ABB RobotStudio station: roboticcell.rsstnx

Station roboticcell (saved by RobotStudio 23.2.10395.0)
Controller Controller2
  mechanical unit ROB_1: IRB2600_20_165_C_01_2, 6 joints, base frame (0, 0, 0) mm
Layout (positions relative to the parent item):
  - IRB2600_20_165_C_01_2 [mechanism, from %ABB.RobotStudio.Models.IRB2600%\IRB2600_20_165_C_01.rslib] at (0, 0, 0) mm; joint values [0.1279, 0.0673, -0.394, 2.9455, -0.603, -2.0324] (rad or m)
  - 2FGP20_WEB_26012022_3 [graphiccomponentgroup] at (0, 0, 0) mm, rotated rx 0 ry 0 rz 90 deg
    - 108791 [graphiccomponentgroup] at (0, 153, -120.5) mm, rotated rx 90 ry 0 rz 180 deg
      - 108659 [graphiccomponentgroup] at (205, 123, 11.8) mm, rotated rx 90 ry 0 rz 24.4 deg
        - 108790 [part] at (0, 0, 0) mm, rotated rx 180 ry 0 rz 0 deg, size 17 x 14.6 x 17 mm
        - 101019 [part] at (0, -6.3, 0) mm, rotated rx 180 ry 74.5 rz 0 deg, size 40 x 26 x 40 mm
        - 104702_Standard [part] at (0, -27.2, 0) mm, rotated rx 90 ry -9.84 rz 180 deg, size 23.8 x 13 x 23.4 mm
        - 109120 [part] at (0, -11.45, 0) mm, rotated rx 180 ry -25.08 rz 0 deg, size 12.6 x 1.3 x 12.6 mm
      - 108659-1 [graphiccomponentgroup] at (-205, 123, 11.8) mm, rotated rx 90 ry 0 rz 137.17 deg
        - 108790 [part] at (0, 0, 0) mm, rotated rx 180 ry 0 rz 0 deg, size 17 x 14.6 x 17 mm
        - 101019 [part] at (0, -6.3, 0) mm, rotated rx 180 ry 74.5 rz 0 deg, size 40 x 26 x 40 mm
        - 104702_Standard [part] at (0, -27.2, 0) mm, rotated rx 90 ry -9.84 rz 180 deg, size 23.8 x 13 x 23.4 mm
        - 109120 [part] at (0, -11.45, 0) mm, rotated rx 180 ry -25.08 rz 0 deg, size 12.6 x 1.3 x 12.6 mm
      - 108659-2 [graphiccomponentgroup] at (205, 8.5, 11.8) mm, rotated rx 90 ry 0 rz -12.46 deg
        - 108790 [part] at (0, 0, 0) mm, rotated rx 180 ry 0 rz 0 deg, size 17 x 14.6 x 17 mm
        - 101019 [part] at (0, -6.3, 0) mm, rotated rx 180 ry 74.5 rz 0 deg, size 40 x 26 x 40 mm
        - 104702_Standard [part] at (0, -27.2, 0) mm, rotated rx 90 ry -9.84 rz 180 deg, size 23.8 x 13 x 23.4 mm
        - 109120 [part] at (0, -11.45, 0) mm, rotated rx 180 ry -25.08 rz 0 deg, size 12.6 x 1.3 x 12.6 mm
      - 108659-3 [graphiccomponentgroup] at (-205, 8.5, 11.8) mm, rotated rx 90 ry 0 rz 173.2 deg
        - 108790 [part] at (0, 0, 0) mm, rotated rx 180 ry 0 rz 0 deg, size 17 x 14.6 x 17 mm
        - 101019 [part] at (0, -6.3, 0) mm, rotated rx 180 ry 74.5 rz 0 deg, size 40 x 26 x 40 mm
        - 104702_Standard [part] at (0, -27.2, 0) mm, rotated rx 90 ry -9.84 rz 180 deg, size 23.8 x 13 x 23.4 mm
        - 109120 [part] at (0, -11.45, 0) mm, rotated rx 180 ry -25.08 rz 0 deg, size 12.6 x 1.3 x 12.6 mm
      - 101014 [part] at (-75, 38, 4.4) mm, rotated rx 0 ry 90 rz 50.35 deg, size 14.4 x 9.9 x 10 mm
      - 101014 [part] at (-11, 45, 4.4) mm, rotated rx 0 ry 90 rz 50.35 deg, size 14.4 x 9.9 x 10 mm
      - 108792 [part] at (0, 30, 0) mm, rotated rx -90 ry 0 rz 180 deg, size 427 x 3 x 101.5 mm
      - 109119_Right version [part] at (101.22, 54.39, 10.55) mm, rotated rx -93.67 ry 0 rz 34.23 deg, size 171.2 x 32 x 18.8 mm
      - 109119 [part] at (-101.34, 54.21, 10.57) mm, rotated rx -92.75 ry 0 rz 147.01 deg, size 171.2 x 32 x 18.8 mm
      - 101014 [part] at (11, 45, 4.4) mm, rotated rx 0 ry 90 rz -50.35 deg, size 14.4 x 9.9 x 10 mm
      - 101014 [part] at (75, 38, 4.4) mm, rotated rx 0 ry 90 rz -50.35 deg, size 14.4 x 9.9 x 10 mm
      - 101014 [part] at (-75, 16, 4.4) mm, rotated rx 0 ry 90 rz 44.86 deg, size 14.4 x 9.9 x 10 mm
      - 108793 [part] at (0, 0, 0) mm, rotated rx -90 ry 0 rz 180 deg, size 427 x 3 x 29 mm
      - 109118 [part] at (200.6, 8.7, -15.4) mm, rotated rx 93.46 ry 0 rz 177.37 deg, size 150 x 32 x 6 mm
      - 109118 [part] at (-200.6, 8.7, -15.4) mm, rotated rx 86.54 ry 0 rz 2.63 deg, size 150 x 32 x 6 mm
      - 101014 [part] at (75, 16, 4.4) mm, rotated rx 0 ry 90 rz -44.86 deg, size 14.4 x 9.9 x 10 mm
      - 104702_Standard [part] at (-41, 16, 9.4) mm, rotated rx 180 ry 0 rz 180 deg, size 23.8 x 13 x 23.4 mm
      - 104702_Standard [part] at (-41, 38, 9.4) mm, rotated rx 180 ry 0 rz 180 deg, size 23.8 x 13 x 23.4 mm
      - 104702_Standard [part] at (41, 16, 9.4) mm, rotated rx 180 ry 0 rz 0 deg, size 23.8 x 13 x 23.4 mm
      - 104702_Standard [part] at (41, 38, 9.4) mm, rotated rx 180 ry 0 rz 0 deg, size 23.8 x 13 x 23.4 mm
    - Base [graphiccomponentgroup] at (0, 0, 0) mm, rotated rx 0 ry 0 rz -90 deg
      - 109304 [part] at (50, 0, -120.5) mm, rotated rx 90 ry 0 rz 180 deg, size 400 x 78 x 188 mm
      - 109120 [part] at (-17.68, -17.68, -42.95) mm, rotated rx 90 ry 0 rz -90 deg, size 12.6 x 1.3 x 12.6 mm
      - 109120 [part] at (-17.68, 17.68, -42.95) mm, rotated rx 90 ry 0 rz -90 deg, size 12.6 x 1.3 x 12.6 mm
      - 109120 [part] at (17.68, 17.68, -42.95) mm, rotated rx 90 ry 0 rz -90 deg, size 12.6 x 1.3 x 12.6 mm
      - 109120 [part] at (17.68, -17.68, -42.95) mm, rotated rx 90 ry 0 rz -90 deg, size 12.6 x 1.3 x 12.6 mm
      - 108732 [graphiccomponentgroup] at (0, 0, -112.5) mm, rotated rx 90 ry 0 rz -90 deg
        - 107607 [part], size 187.8 x 85.2 x 399.8 mm
        - 108733 [part] at (-17.68, 70, 17.68) mm, rotated rx -90 ry 1.86 rz 0 deg, size 10 x 10 x 29.7 mm
        - 108733 [part] at (-17.68, 70, -17.68) mm, rotated rx -90 ry 1.86 rz 0 deg, size 10 x 10 x 29.7 mm
        - 108733 [part] at (17.68, 99.7, -17.68) mm, rotated rx -90 ry 1.86 rz 180 deg, size 10 x 10 x 29.7 mm
        - 108733 [part] at (17.68, 99.7, 17.68) mm, rotated rx -90 ry 1.86 rz 180 deg, size 10 x 10 x 29.7 mm
      - 108677_Bended [part] at (0, 0, -112.5) mm, rotated rx 90 ry 0 rz -90 deg, size 187.4 x 41.4 x 399.9 mm
      - 104110 [graphiccomponentgroup] at (55.39, -142.12, 182.44) mm, rotated rx -90 ry 0 rz 180 deg
        - 101144 [graphiccomponentgroup] at (70.12, 187.24, -146.12) mm, rotated rx 180 ry 0 rz 0 deg
          - 101145 [part], size 6 x 2.8 x 4 mm
          - 101146 [part] at (0.77, -3.58, -1) mm, rotated rx 3.05 ry 0 rz 90 deg, size 3.9 x 1.7 x 1.7 mm
          - 101147 [part] at (0.77, -1.94, -1) mm, rotated rx 5.39 ry 0 rz 90 deg, size 3.4 x 1 x 1 mm
          - 101148 [part] at (0.77, -3.58, -1) mm, rotated rx 180 ry 0 rz 90 deg, size 2.6 x 1 x 1.1 mm
          - 101149 [part] at (0.77, -2.72, -1) mm, rotated rx -90 ry -11.12 rz 0 deg, size 0.8 x 0.8 x 3.5 mm
          - 101149 [part] at (0.77, -2.72, -3) mm, rotated rx -90 ry -11.12 rz 0 deg, size 0.8 x 0.8 x 3.5 mm
          - 101148 [part] at (0.77, -3.58, -3) mm, rotated rx 180 ry 0 rz 90 deg, size 2.6 x 1 x 1.1 mm
          - 101147 [part] at (0.77, -1.94, -3) mm, rotated rx -61.01 ry 0 rz 90 deg, size 3.4 x 1 x 1 mm
          - 101146 [part] at (0.77, -3.58, -3) mm, rotated rx 0 ry 0 rz 90 deg, size 3.9 x 1.7 x 1.7 mm
          - 101149 [part] at (2.77, -2.72, -1) mm, rotated rx -90 ry -11.12 rz 0 deg, size 0.8 x 0.8 x 3.5 mm
          - 101149 [part] at (2.77, -2.72, -3) mm, rotated rx -90 ry -11.12 rz 0 deg, size 0.8 x 0.8 x 3.5 mm
          - 101148 [part] at (2.77, -3.58, -1) mm, rotated rx 180 ry 0 rz 90 deg, size 2.6 x 1 x 1.1 mm
          - 101148 [part] at (2.77, -3.58, -3) mm, rotated rx 180 ry 0 rz 90 deg, size 2.6 x 1 x 1.1 mm
          - 101147 [part] at (2.77, -1.94, -1) mm, rotated rx 180 ry 0 rz 90 deg, size 3.4 x 1 x 1 mm
          - 101147 [part] at (2.77, -1.94, -3) mm, rotated rx 163.02 ry 0 rz 90 deg, size 3.4 x 1 x 1 mm
          - 101146 [part] at (2.77, -3.58, -1) mm, rotated rx 0 ry 0 rz 90 deg, size 3.9 x 1.7 x 1.7 mm
          - 101146 [part] at (2.77, -3.58, -3) mm, rotated rx 0 ry 0 rz 90 deg, size 3.9 x 1.7 x 1.7 mm
          - 101149 [part] at (4.77, -2.72, -1) mm, rotated rx -90 ry -11.12 rz 0 deg, size 0.8 x 0.8 x 3.5 mm
          - 101149 [part] at (4.77, -2.72, -3) mm, rotated rx -90 ry -11.12 rz 0 deg, size 0.8 x 0.8 x 3.5 mm
          - 101148 [part] at (4.77, -3.58, -1) mm, rotated rx 180 ry 0 rz 90 deg, size 2.6 x 1 x 1.1 mm
          - 101148 [part] at (4.77, -3.58, -3) mm, rotated rx 180 ry 0 rz 90 deg, size 2.6 x 1 x 1.1 mm
          - 101147 [part] at (4.77, -1.94, -1) mm, rotated rx 180 ry 0 rz 90 deg, size 3.4 x 1 x 1 mm
          - 101147 [part] at (4.77, -1.94, -3) mm, rotated rx 180 ry 0 rz 90 deg, size 3.4 x 1 x 1 mm
          - 101146 [part] at (4.77, -3.58, -1) mm, rotated rx 0 ry 0 rz 90 deg, size 3.9 x 1.7 x 1.7 mm
          - 101146 [part] at (4.77, -3.58, -3) mm, rotated rx 0 ry 0 rz 90 deg, size 3.9 x 1.7 x 1.7 mm
        - 101144-1 [graphiccomponentgroup] at (75.65, 187.24, -138.12) mm, rotated rx 0 ry 0 rz 180 deg
          - 101145 [part], size 6 x 2.8 x 4 mm
          - 101146 [part] at (0.77, -3.58, -1) mm, rotated rx 3.05 ry 0 rz 90 deg, size 3.9 x 1.7 x 1.7 mm
          - 101147 [part] at (0.77, -1.94, -1) mm, rotated rx 5.39 ry 0 rz 90 deg, size 3.4 x 1 x 1 mm
          - 101148 [part] at (0.77, -3.58, -1) mm, rotated rx 180 ry 0 rz 90 deg, size 2.6 x 1 x 1.1 mm
          - 101149 [part] at (0.77, -2.72, -1) mm, rotated rx -90 ry -11.12 rz 0 deg, size 0.8 x 0.8 x 3.5 mm
          - 101149 [part] at (0.77, -2.72, -3) mm, rotated rx -90 ry -11.12 rz 0 deg, size 0.8 x 0.8 x 3.5 mm
          - 101148 [part] at (0.77, -3.58, -3) mm, rotated rx 180 ry 0 rz 90 deg, size 2.6 x 1 x 1.1 mm
          - 101147 [part] at (0.77, -1.94, -3) mm, rotated rx -61.01 ry 0 rz 90 deg, size 3.4 x 1 x 1 mm
          - 101146 [part] at (0.77, -3.58, -3) mm, rotated rx 0 ry 0 rz 90 deg, size 3.9 x 1.7 x 1.7 mm
          - 101149 [part] at (2.77, -2.72, -1) mm, rotated rx -90 ry -11.12 rz 0 deg, size 0.8 x 0.8 x 3.5 mm
          - 101149 [part] at (2.77, -2.72, -3) mm, rotated rx -90 ry -11.12 rz 0 deg, size 0.8 x 0.8 x 3.5 mm
          - 101148 [part] at (2.77, -3.58, -1) mm, rotated rx 180 ry 0 rz 90 deg, size 2.6 x 1 x 1.1 mm
          - 101148 [part] at (2.77, -3.58, -3) mm, rotated rx 180 ry 0 rz 90 deg, size 2.6 x 1 x 1.1 mm
          - 101147 [part] at (2.77, -1.94, -1) mm, rotated rx 180 ry 0 rz 90 deg, size 3.4 x 1 x 1 mm
          - 101147 [part] at (2.77, -1.94, -3) mm, rotated rx 163.02 ry 0 rz 90 deg, size 3.4 x 1 x 1 mm
          - 101146 [part] at (2.77, -3.58, -1) mm, rotated rx 0 ry 0 rz 90 deg, size 3.9 x 1.7 x 1.7 mm
          - 101146 [part] at (2.77, -3.58, -3) mm, rotated rx 0 ry 0 rz 90 deg, size 3.9 x 1.7 x 1.7 mm
          - 101149 [part] at (4.77, -2.72, -1) mm, rotated rx -90 ry -11.12 rz 0 deg, size 0.8 x 0.8 x 3.5 mm
          - 101149 [part] at (4.77, -2.72, -3) mm, rotated rx -90 ry -11.12 rz 0 deg, size 0.8 x 0.8 x 3.5 mm
          - 101148 [part] at (4.77, -3.58, -1) mm, rotated rx 180 ry 0 rz 90 deg, size 2.6 x 1 x 1.1 mm
          - 101148 [part] at (4.77, -3.58, -3) mm, rotated rx 180 ry 0 rz 90 deg, size 2.6 x 1 x 1.1 mm
          - 101147 [part] at (4.77, -1.94, -1) mm, rotated rx 180 ry 0 rz 90 deg, size 3.4 x 1 x 1 mm
          - 101147 [part] at (4.77, -1.94, -3) mm, rotated rx 180 ry 0 rz 90 deg, size 3.4 x 1 x 1 mm
          - 101146 [part] at (4.77, -3.58, -1) mm, rotated rx 0 ry 0 rz 90 deg, size 3.9 x 1.7 x 1.7 mm
          - 101146 [part] at (4.77, -3.58, -3) mm, rotated rx 0 ry 0 rz 90 deg, size 3.9 x 1.7 x 1.7 mm
        - 101164 [part] at (55.39, 192.94, -142.12) mm, size 70.6 x 4 x 71 mm
        - 102785 [part] at (55.39, 181.74, -142.12) mm, rotated rx 0 ry -90 rz -180 deg, size 60.6 x 11.2 x 65.9 mm
        - 102784 [part] at (55.39, 187.79, -103.32) mm, rotated rx 0 ry 90 rz 0 deg, size 20.6 x 7.5 x 31.8 mm
        - 101386 [part] at (72.89, 189.32, -142.12) mm, rotated rx 0 ry -90 rz -180 deg, size 12 x 4.3 x 10 mm
        - 101014 [part] at (73.07, 186.14, -124.44) mm, rotated rx 116.38 ry 0 rz 90 deg, size 14.4 x 9.9 x 10 mm
        - 101014 [part] at (37.71, 186.14, -124.44) mm, rotated rx -53.18 ry 0 rz 90 deg, size 14.4 x 9.9 x 10 mm
        - 101014 [part] at (73.07, 186.14, -159.79) mm, rotated rx -53.18 ry 0 rz 90 deg, size 14.4 x 9.9 x 10 mm
        - 101014 [part] at (37.71, 186.14, -159.79) mm, rotated rx -53.18 ry 0 rz 90 deg, size 14.4 x 9.9 x 10 mm
      - 103927 [part] at (142.67, 0, -35.5) mm, rotated rx 11.95 ry 0 rz 90 deg, size 22.7 x 24.6 x 0.2 mm
      - 100142 [part] at (-151.2, -41, -104.5) mm, rotated rx 0 ry 60 rz -90 deg, size 14 x 6.8 x 15 mm
      - 100142 [part] at (-151.2, -41, -82.5) mm, rotated rx 0 ry 60 rz -90 deg, size 14 x 6.8 x 15 mm
      - 100142 [part] at (-151.2, 41, -82.5) mm, rotated rx 0 ry 60 rz -90 deg, size 14 x 6.8 x 15 mm
    - Finger [graphiccomponentgroup] at (0, 0, 0) mm, rotated rx 0 ry 0 rz -90 deg
      - 108692 [part] at (-120.5, 0, -132.1) mm, rotated rx 90 ry 0 rz 90 deg, size 185 x 11.6 x 56 mm
      - 109273 [graphiccomponentgroup] at (-92.5, 0, -132.1) mm, rotated rx 0 ry 0 rz 180 deg
        - 108713 [part], size 80.8 x 186 x 220 mm
        - 108801 [part] at (75.75, 0, -194.9) mm, rotated rx 180 ry 0 rz -90 deg, size 186 x 6 x 50 mm
        - 101722 [part] at (80.75, -68, -208.5) mm, rotated rx 0 ry 62.4 rz -90 deg, size 8.4 x 8 x 8.4 mm
        - 101722 [part] at (80.75, 68, -208.5) mm, rotated rx 0 ry 47.55 rz -90 deg, size 8.4 x 8 x 8.4 mm
        - 108801 [part] at (75.75, 0, -86.1) mm, rotated rx 0 ry 0 rz 90 deg, size 186 x 6 x 50 mm
        - 101722 [part] at (80.75, 68, -181.3) mm, rotated rx 0 ry 47.55 rz -90 deg, size 8.4 x 8 x 8.4 mm
        - 101722 [part] at (80.75, -68, -181.3) mm, rotated rx 0 ry 62.4 rz -90 deg, size 8.4 x 8 x 8.4 mm
        - 101722 [part] at (80.75, 68, -99.7) mm, rotated rx 0 ry 47.55 rz -90 deg, size 8.4 x 8 x 8.4 mm
        - 101722 [part] at (80.75, 68, -72.5) mm, rotated rx 0 ry 47.55 rz -90 deg, size 8.4 x 8 x 8.4 mm
        - 101722 [part] at (80.75, -68, -99.7) mm, rotated rx 0 ry 62.4 rz -90 deg, size 8.4 x 8 x 8.4 mm
        - 101722 [part] at (80.75, -68, -72.5) mm, rotated rx 0 ry 62.4 rz -90 deg, size 8.4 x 8 x 8.4 mm
      - 108686 [part] at (-141.5, 0, -137.1) mm, rotated rx -90 ry 0 rz 89.62 deg, size 11.3 x 12 x 11.3 mm
      - 108686 [part] at (-99.5, 0, -137.1) mm, rotated rx -90 ry 0 rz 89.62 deg, size 11.3 x 12 x 11.3 mm
      - 108686 [part] at (-141.5, -65, -137.1) mm, rotated rx -90 ry 0 rz 89.62 deg, size 11.3 x 12 x 11.3 mm
      - 108686 [part] at (-99.5, -65, -137.1) mm, rotated rx -90 ry 0 rz 89.62 deg, size 11.3 x 12 x 11.3 mm
      - 108686 [part] at (-141.5, 65, -137.1) mm, rotated rx -90 ry 0 rz 89.62 deg, size 11.3 x 12 x 11.3 mm
      - 108686 [part] at (-99.5, 65, -137.1) mm, rotated rx -90 ry 0 rz 89.62 deg, size 11.3 x 12 x 11.3 mm
      - 102333 [part] at (-129.46, 86, -131.9) mm, rotated rx 0 ry -90 rz 125.83 deg, size 16.4 x 10 x 10 mm
      - 102333 [part] at (-107.46, 86, -131.9) mm, rotated rx 0 ry -90 rz 125.83 deg, size 16.4 x 10 x 10 mm
      - 102333 [part] at (-107.46, -86, -131.9) mm, rotated rx 0 ry -90 rz 125.83 deg, size 16.4 x 10 x 10 mm
      - 102333 [part] at (-129.46, -86, -131.9) mm, rotated rx 0 ry -90 rz 125.83 deg, size 16.4 x 10 x 10 mm
      - 100142 [part] at (-151.2, 41, -104.5) mm, rotated rx 0 ry 60 rz -90 deg, size 14 x 6.8 x 15 mm
    - Moving_Finger [graphiccomponentgroup] at (0, 0, 0) mm, rotated rx 0 ry 0 rz -90 deg
      - 109273-1 [graphiccomponentgroup] at (192.5, 0, -132.1) mm
        - 108713 [part], size 80.8 x 186 x 220 mm
        - 108801 [part] at (75.75, 0, -194.9) mm, rotated rx 180 ry 0 rz -90 deg, size 186 x 6 x 50 mm
        - 101722 [part] at (80.75, -68, -208.5) mm, rotated rx 0 ry 62.4 rz -90 deg, size 8.4 x 8 x 8.4 mm
        - 101722 [part] at (80.75, 68, -208.5) mm, rotated rx 0 ry 47.55 rz -90 deg, size 8.4 x 8 x 8.4 mm
        - 108801 [part] at (75.75, 0, -86.1) mm, rotated rx 0 ry 0 rz 90 deg, size 186 x 6 x 50 mm
        - 101722 [part] at (80.75, 68, -181.3) mm, rotated rx 0 ry 47.55 rz -90 deg, size 8.4 x 8 x 8.4 mm
        - 101722 [part] at (80.75, -68, -181.3) mm, rotated rx 0 ry 62.4 rz -90 deg, size 8.4 x 8 x 8.4 mm
        - 101722 [part] at (80.75, 68, -99.7) mm, rotated rx 0 ry 47.55 rz -90 deg, size 8.4 x 8 x 8.4 mm
        - 101722 [part] at (80.75, 68, -72.5) mm, rotated rx 0 ry 47.55 rz -90 deg, size 8.4 x 8 x 8.4 mm
        - 101722 [part] at (80.75, -68, -99.7) mm, rotated rx 0 ry 62.4 rz -90 deg, size 8.4 x 8 x 8.4 mm
        - 101722 [part] at (80.75, -68, -72.5) mm, rotated rx 0 ry 62.4 rz -90 deg, size 8.4 x 8 x 8.4 mm
      - 108686 [part] at (241.5, 0, -137.1) mm, rotated rx -90 ry 0 rz 177.92 deg, size 11.3 x 12 x 11.3 mm
      - 108686 [part] at (199.5, 0, -137.1) mm, rotated rx -90 ry 0 rz 177.92 deg, size 11.3 x 12 x 11.3 mm
      - 108686 [part] at (241.5, 65, -137.1) mm, rotated rx -90 ry 0 rz 177.92 deg, size 11.3 x 12 x 11.3 mm
      - 108686 [part] at (199.5, 65, -137.1) mm, rotated rx -90 ry 0 rz 177.92 deg, size 11.3 x 12 x 11.3 mm
      - 108686 [part] at (241.5, -65, -137.1) mm, rotated rx -90 ry 0 rz 177.92 deg, size 11.3 x 12 x 11.3 mm
      - 108686 [part] at (199.5, -65, -137.1) mm, rotated rx -90 ry 0 rz 177.92 deg, size 11.3 x 12 x 11.3 mm
      - 107611 [part] at (220.5, 0, -132.1) mm, rotated rx 90 ry 0 rz -90 deg, size 185 x 11 x 56 mm
      - 107216 [part] at (214.5, -75, -128.25) mm, rotated rx 0 ry -90 rz 113.11 deg, size 13.7 x 8.4 x 8.5 mm
      - 107216 [part] at (214.5, 75, -128.25) mm, rotated rx 0 ry -90 rz 113.11 deg, size 13.7 x 8.4 x 8.5 mm
      - 107216 [part] at (229.5, 75, -128.25) mm, rotated rx 0 ry -90 rz 113.11 deg, size 13.7 x 8.4 x 8.5 mm
      - 107216 [part] at (199.5, 75, -128.25) mm, rotated rx 0 ry -90 rz 113.11 deg, size 13.7 x 8.4 x 8.5 mm
      - 107216 [part] at (229.5, -75, -128.25) mm, rotated rx 0 ry -90 rz 113.11 deg, size 13.7 x 8.4 x 8.5 mm
      - 107216 [part] at (199.5, -75, -128.25) mm, rotated rx 0 ry -90 rz 113.11 deg, size 13.7 x 8.4 x 8.5 mm
  - Conveyor_400 [smart component, from Feeders\Conveyor_400.rslib] at (1000, -200, 0) mm
      properties: PreparationTime_ToPick=0; Product_ToPick=; ClearTime_Placed=0; Product_Placed=
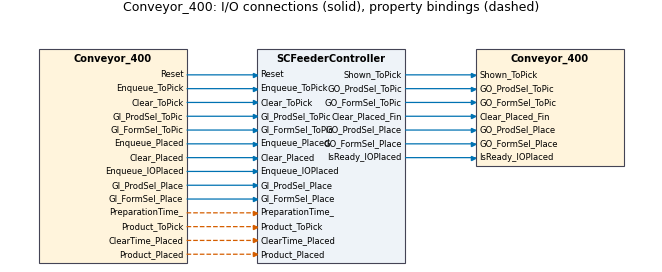
      connections:
        Conveyor_400.Reset -> SCFeederController.Reset
        Conveyor_400.Enqueue_ToPick -> SCFeederController.Enqueue_ToPick
        SCFeederController.Shown_ToPick -> Conveyor_400.Shown_ToPick
        Conveyor_400.Clear_ToPick -> SCFeederController.Clear_ToPick
        Conveyor_400.GI_ProdSel_ToPick -> SCFeederController.GI_ProdSel_ToPick
        Conveyor_400.GI_FormSel_ToPick -> SCFeederController.GI_FormSel_ToPick
        SCFeederController.GO_ProdSel_ToPick -> Conveyor_400.GO_ProdSel_ToPick
        SCFeederController.GO_FormSel_ToPick -> Conveyor_400.GO_FormSel_ToPick
        SCFeederController.Clear_Placed_Finished -> Conveyor_400.Clear_Placed_Finished
        Conveyor_400.Enqueue_Placed -> SCFeederController.Enqueue_Placed
        Conveyor_400.Clear_Placed -> SCFeederController.Clear_Placed
        Conveyor_400.Enqueue_IOPlacedRequest -> SCFeederController.Enqueue_IOPlacedRequest
        Conveyor_400.GI_ProdSel_PlacedRequest -> SCFeederController.GI_ProdSel_PlacedRequest
        Conveyor_400.GI_FormSel_PlacedRequest -> SCFeederController.GI_FormSel_PlacedRequest
        SCFeederController.GO_ProdSel_PlacedRequest -> Conveyor_400.GO_ProdSel_PlacedRequest
        SCFeederController.GO_FormSel_PlacedRequest -> Conveyor_400.GO_FormSel_PlacedRequest
        SCFeederController.IsReady_IOPlacedRequest -> Conveyor_400.IsReady_IOPlacedRequest
        Conveyor_400.PreparationTime_ToPick => SCFeederController.PreparationTime_ToPick
        Conveyor_400.Product_ToPick => SCFeederController.Product_ToPick
        Conveyor_400.ClearTime_Placed => SCFeederController.ClearTime_Placed
        Conveyor_400.Product_Placed => SCFeederController.Product_Placed
    - 400_guide [part, from Feeders\Conveyor_400.rslib]
    - SCFeederController [smart component, from Components\SC_FeederController.rslib]
        properties: Product_Placed=; ClearTime_Placed=0; PreparationTime_ToPick=0; Product_ToPick=
  - Conveyor_1200_with Pallet [smart component, from Feeders\Conveyor_1200_with Pallet.rslib] at (-561.25, -2004.97, 0) mm
      properties: PreparationTime_ToPick=0; Product_ToPick=; ClearTime_Placed=0; Product_Placed=
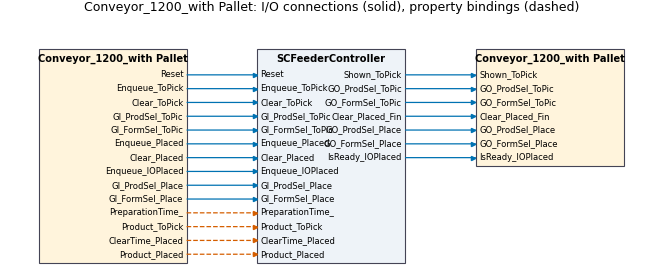
      connections:
        Conveyor_1200_with Pallet.Reset -> SCFeederController.Reset
        Conveyor_1200_with Pallet.Enqueue_ToPick -> SCFeederController.Enqueue_ToPick
        SCFeederController.Shown_ToPick -> Conveyor_1200_with Pallet.Shown_ToPick
        Conveyor_1200_with Pallet.Clear_ToPick -> SCFeederController.Clear_ToPick
        Conveyor_1200_with Pallet.GI_ProdSel_ToPick -> SCFeederController.GI_ProdSel_ToPick
        Conveyor_1200_with Pallet.GI_FormSel_ToPick -> SCFeederController.GI_FormSel_ToPick
        SCFeederController.GO_ProdSel_ToPick -> Conveyor_1200_with Pallet.GO_ProdSel_ToPick
        SCFeederController.GO_FormSel_ToPick -> Conveyor_1200_with Pallet.GO_FormSel_ToPick
        SCFeederController.Clear_Placed_Finished -> Conveyor_1200_with Pallet.Clear_Placed_Finished
        Conveyor_1200_with Pallet.Enqueue_Placed -> SCFeederController.Enqueue_Placed
        Conveyor_1200_with Pallet.Clear_Placed -> SCFeederController.Clear_Placed
        Conveyor_1200_with Pallet.Enqueue_IOPlacedRequest -> SCFeederController.Enqueue_IOPlacedRequest
        Conveyor_1200_with Pallet.GI_ProdSel_PlacedRequest -> SCFeederController.GI_ProdSel_PlacedRequest
        Conveyor_1200_with Pallet.GI_FormSel_PlacedRequest -> SCFeederController.GI_FormSel_PlacedRequest
        SCFeederController.GO_ProdSel_PlacedRequest -> Conveyor_1200_with Pallet.GO_ProdSel_PlacedRequest
        SCFeederController.GO_FormSel_PlacedRequest -> Conveyor_1200_with Pallet.GO_FormSel_PlacedRequest
        SCFeederController.IsReady_IOPlacedRequest -> Conveyor_1200_with Pallet.IsReady_IOPlacedRequest
        Conveyor_1200_with Pallet.PreparationTime_ToPick => SCFeederController.PreparationTime_ToPick
        Conveyor_1200_with Pallet.Product_ToPick => SCFeederController.Product_ToPick
        Conveyor_1200_with Pallet.ClearTime_Placed => SCFeederController.ClearTime_Placed
        Conveyor_1200_with Pallet.Product_Placed => SCFeederController.Product_Placed
    - Conv_Pallet [graphiccomponentgroup, from Feeders\Conveyor_1200_with Pallet.rslib]
      - Conv_950_4000 [part, from Feeders\Conveyor_1200_with Pallet.rslib]
      - DWPallet [part, from Feeders\Conveyor_1200_with Pallet.rslib] at (60, 4.38, 413.27) mm
    - SCFeederController [smart component, from Components\SC_FeederController.rslib]
        properties: Product_Placed=; ClearTime_Placed=0; PreparationTime_ToPick=0; Product_ToPick=
  - Conveyor_1200_with Pallet_1 [smart component, from Feeders\Conveyor_1200_with Pallet.rslib] at (-561.25, 995.03, 0) mm
      properties: PreparationTime_ToPick=0; Product_ToPick=; ClearTime_Placed=0; Product_Placed=
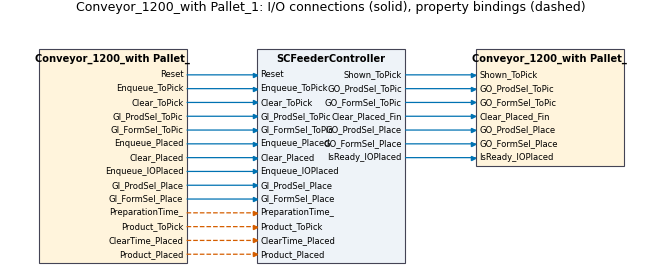
      connections:
        Conveyor_1200_with Pallet_1.Reset -> SCFeederController.Reset
        Conveyor_1200_with Pallet_1.Enqueue_ToPick -> SCFeederController.Enqueue_ToPick
        SCFeederController.Shown_ToPick -> Conveyor_1200_with Pallet_1.Shown_ToPick
        Conveyor_1200_with Pallet_1.Clear_ToPick -> SCFeederController.Clear_ToPick
        Conveyor_1200_with Pallet_1.GI_ProdSel_ToPick -> SCFeederController.GI_ProdSel_ToPick
        Conveyor_1200_with Pallet_1.GI_FormSel_ToPick -> SCFeederController.GI_FormSel_ToPick
        SCFeederController.GO_ProdSel_ToPick -> Conveyor_1200_with Pallet_1.GO_ProdSel_ToPick
        SCFeederController.GO_FormSel_ToPick -> Conveyor_1200_with Pallet_1.GO_FormSel_ToPick
        SCFeederController.Clear_Placed_Finished -> Conveyor_1200_with Pallet_1.Clear_Placed_Finished
        Conveyor_1200_with Pallet_1.Enqueue_Placed -> SCFeederController.Enqueue_Placed
        Conveyor_1200_with Pallet_1.Clear_Placed -> SCFeederController.Clear_Placed
        Conveyor_1200_with Pallet_1.Enqueue_IOPlacedRequest -> SCFeederController.Enqueue_IOPlacedRequest
        Conveyor_1200_with Pallet_1.GI_ProdSel_PlacedRequest -> SCFeederController.GI_ProdSel_PlacedRequest
        Conveyor_1200_with Pallet_1.GI_FormSel_PlacedRequest -> SCFeederController.GI_FormSel_PlacedRequest
        SCFeederController.GO_ProdSel_PlacedRequest -> Conveyor_1200_with Pallet_1.GO_ProdSel_PlacedRequest
        SCFeederController.GO_FormSel_PlacedRequest -> Conveyor_1200_with Pallet_1.GO_FormSel_PlacedRequest
        SCFeederController.IsReady_IOPlacedRequest -> Conveyor_1200_with Pallet_1.IsReady_IOPlacedRequest
        Conveyor_1200_with Pallet_1.PreparationTime_ToPick => SCFeederController.PreparationTime_ToPick
        Conveyor_1200_with Pallet_1.Product_ToPick => SCFeederController.Product_ToPick
        Conveyor_1200_with Pallet_1.ClearTime_Placed => SCFeederController.ClearTime_Placed
        Conveyor_1200_with Pallet_1.Product_Placed => SCFeederController.Product_Placed
    - Conv_Pallet [graphiccomponentgroup, from Feeders\Conveyor_1200_with Pallet.rslib]
      - Conv_950_4000 [part, from Feeders\Conveyor_1200_with Pallet.rslib]
      - DWPallet [part, from Feeders\Conveyor_1200_with Pallet.rslib] at (60, 4.38, 413.27) mm
    - SCFeederController [smart component, from Components\SC_FeederController.rslib]
        properties: Product_Placed=; ClearTime_Placed=0; PreparationTime_ToPick=0; Product_ToPick=
  - Gripper [smart component, from Components\GripperOR.rslib] at (987.7, 117.57, 1485.12) mm, rotated rx -65.9 ry -49.98 rz 71.85 deg
      properties: ReleasedObject=(none)
    - Gripper [mechanism] at (0, 0, 0) mm; joint values [-0.012] (rad or m)
        TCP Gripper at (-162.25, 0.02, -218.2) mm
        links: Base, Finger, MovingFinger, Ventosa
    - Clamp1 [smart component]
      - ClampControl [smart component]
  - PalletPattern1 [graphiccomponentgroup] at (700, -1200, 557.91) mm, rotated rx 0 ry 0 rz 180 deg
  - Frame_5 [frame] at (-162.25, 0.02, -218.2) mm, rotated rx 180 ry 0 rz 90 deg
Attachment: pmInfeeder1_WObj is attached to Conveyor_400
Attachment: pmOutfeeder3_WObj is attached to Conveyor_1200_with Pallet
Attachment: pmOutfeeder1_WObj is attached to Conveyor_1200_with Pallet_1
Attachment: Gripper is attached to IRB2600_20_165_C_01_2 / Link6
Targets, tools, work objects and paths stored in the station, written as RAPID:
! task T_ROB1
MODULE pmrcUser
  TASK PERS wobjdata pmInfeeder1_WObj:=[FALSE,TRUE,"",[[0,0,0],[1,0,0,0]],[[0,0,0],[1,0,0,0]]];
  TASK PERS wobjdata pmInfeeder2_WObj:=[FALSE,TRUE,"",[[0,0,0],[1,0,0,0]],[[0,0,0],[1,0,0,0]]];
  TASK PERS wobjdata pmInfeeder3_WObj:=[FALSE,TRUE,"",[[0,0,0],[1,0,0,0]],[[0,0,0],[1,0,0,0]]];
  TASK PERS wobjdata pmInfeeder4_WObj:=[FALSE,TRUE,"",[[0,0,0],[1,0,0,0]],[[0,0,0],[1,0,0,0]]];
  TASK PERS wobjdata pmOutfeeder1_WObj:=[FALSE,TRUE,"",[[0,0,0],[1,0,0,0]],[[0,0,0],[1,0,0,0]]];
  TASK PERS wobjdata pmOutfeeder2_WObj:=[FALSE,TRUE,"",[[0,0,0],[1,0,0,0]],[[0,0,0],[1,0,0,0]]];
  TASK PERS wobjdata pmOutfeeder3_WObj:=[FALSE,TRUE,"",[[0,0,0],[1,0,0,0]],[[0,0,0],[1,0,0,0]]];
  TASK PERS wobjdata pmOutfeeder4_WObj:=[FALSE,TRUE,"",[[0,0,0],[1,0,0,0]],[[0,0,0],[1,0,0,0]]];
  TASK PERS wobjdata pmPallet1_WObj:=[FALSE,TRUE,"",[[0,0,0],[1,0,0,0]],[[0,0,0],[1,0,0,0]]];
  TASK PERS wobjdata pmSlipsheet1_WObj:=[FALSE,TRUE,"",[[0,0,0],[1,0,0,0]],[[0,0,0],[1,0,0,0]]];
  TASK PERS tooldata pmPickTool1:=[TRUE,[[0,0,0],[1,0,0,0]],[1,[0,0,10],[1,0,0,0],0.01,0.01,0.01]];
  TASK PERS tooldata pmSearchTool1:=[TRUE,[[0,0,0],[1,0,0,0]],[1,[0,0,10],[1,0,0,0],0.01,0.01,0.01]];
ENDMODULE

! task T_ROB1
MODULE pmrcSys
  TASK PERS wobjdata pm_home_WObj:=[FALSE,TRUE,"",[[0,0,0],[1,0,0,0]],[[0,0,0],[1,0,0,0]]];
ENDMODULE

! task T_ROB1
MODULE pmrcUser
  TASK PERS wobjdata pmInfeeder1_WObj:=[FALSE,TRUE,"",[[0,0,0],[1,0,0,0]],[[0,0,0],[1,0,0,0]]];
  TASK PERS wobjdata pmInfeeder2_WObj:=[FALSE,TRUE,"",[[0,0,0],[1,0,0,0]],[[0,0,0],[1,0,0,0]]];
  TASK PERS wobjdata pmInfeeder3_WObj:=[FALSE,TRUE,"",[[0,0,0],[1,0,0,0]],[[0,0,0],[1,0,0,0]]];
  TASK PERS wobjdata pmInfeeder4_WObj:=[FALSE,TRUE,"",[[0,0,0],[1,0,0,0]],[[0,0,0],[1,0,0,0]]];
  TASK PERS wobjdata pmOutfeeder1_WObj:=[FALSE,TRUE,"",[[0,0,0],[1,0,0,0]],[[0,0,0],[1,0,0,0]]];
  TASK PERS wobjdata pmOutfeeder2_WObj:=[FALSE,TRUE,"",[[0,0,0],[1,0,0,0]],[[0,0,0],[1,0,0,0]]];
  TASK PERS wobjdata pmOutfeeder3_WObj:=[FALSE,TRUE,"",[[0,0,0],[1,0,0,0]],[[0,0,0],[1,0,0,0]]];
  TASK PERS wobjdata pmOutfeeder4_WObj:=[FALSE,TRUE,"",[[0,0,0],[1,0,0,0]],[[0,0,0],[1,0,0,0]]];
  TASK PERS wobjdata pmPallet1_WObj:=[FALSE,TRUE,"",[[0,0,0],[1,0,0,0]],[[0,0,0],[1,0,0,0]]];
  TASK PERS wobjdata pmSlipsheet1_WObj:=[FALSE,TRUE,"",[[0,0,0],[1,0,0,0]],[[0,0,0],[1,0,0,0]]];
  TASK PERS tooldata pmPickTool1:=[TRUE,[[0,0,0],[1,0,0,0]],[1,[0,0,10],[1,0,0,0],0.01,0.01,0.01]];
  TASK PERS tooldata pmSearchTool1:=[TRUE,[[0,0,0],[1,0,0,0]],[1,[0,0,10],[1,0,0,0],0.01,0.01,0.01]];
ENDMODULE

! task T_ROB1
MODULE pmrcSys
  TASK PERS wobjdata pm_home_WObj:=[FALSE,TRUE,"",[[0,0,0],[1,0,0,0]],[[0,0,0],[1,0,0,0]]];
ENDMODULE

! task T_ROB1
MODULE pmrcUser
  TASK PERS wobjdata pmInfeeder1_WObj:=[FALSE,TRUE,"",[[1000,200,775],[1,0,0,0]],[[0,0,0],[1,0,0,0]]];
  TASK PERS wobjdata pmInfeeder2_WObj:=[FALSE,TRUE,"",[[0,0,0],[1,0,0,0]],[[0,0,0],[1,0,0,0]]];
  TASK PERS wobjdata pmInfeeder3_WObj:=[FALSE,TRUE,"",[[0,0,0],[1,0,0,0]],[[0,0,0],[1,0,0,0]]];
  TASK PERS wobjdata pmInfeeder4_WObj:=[FALSE,TRUE,"",[[0,0,0],[1,0,0,0]],[[0,0,0],[1,0,0,0]]];
  TASK PERS wobjdata pmOutfeeder1_WObj:=[FALSE,TRUE,"",[[-500,1800,557.912],[1,0,0,0]],[[0,0,0],[1,0,0,0]]];
  TASK PERS wobjdata pmOutfeeder2_WObj:=[FALSE,TRUE,"",[[0,0,0],[1,0,0,0]],[[0,0,0],[1,0,0,0]]];
  TASK PERS wobjdata pmOutfeeder3_WObj:=[FALSE,TRUE,"",[[-500,-1200,557.912],[1,0,0,0]],[[0,0,0],[1,0,0,0]]];
  TASK PERS wobjdata pmOutfeeder4_WObj:=[FALSE,TRUE,"",[[0,0,0],[1,0,0,0]],[[0,0,0],[1,0,0,0]]];
  TASK PERS wobjdata pmPallet1_WObj:=[FALSE,TRUE,"",[[0,0,0],[1,0,0,0]],[[0,0,0],[1,0,0,0]]];
  TASK PERS wobjdata pmSlipsheet1_WObj:=[FALSE,TRUE,"",[[0,0,0],[1,0,0,0]],[[0,0,0],[1,0,0,0]]];
  TASK PERS tooldata pmPickTool1:=[TRUE,[[0,0,0],[1,0,0,0]],[0.1,[1092.573,35.885,1174.88],[1,0,0,0],0.000010833,0.000010833,0.000015]];
  TASK PERS tooldata pmSearchTool1:=[TRUE,[[0,0,0],[1,0,0,0]],[0.1,[1092.573,35.885,1174.88],[1,0,0,0],0.000010833,0.000010833,0.000015]];
  TASK PERS tooldata GripperOR:=[TRUE,[[-162.25,0.021,-218.2],[0.707106781,0,0,0.707106781]],[5.34,[1129.958,59.358,1261.756],[1,0,0,0],0.009,0.009,0.009]];
ENDMODULE

! task T_ROB1
MODULE pmrcSys
  TASK PERS wobjdata pm_home_WObj:=[FALSE,TRUE,"",[[0,0,0],[1,0,0,0]],[[0,0,0],[1,0,0,0]]];
ENDMODULE

! task T_ROB1
MODULE CalibData
  PERS tooldata Gripper:=[TRUE,[[-162.25,0.021,-218.2],[1,0,0,0]],[0.1,[1092.573,35.885,1174.88],[1,0,0,0],0,0,0]];
ENDMODULE

